PROGRAM POU
VAR
	
	A : BOOL := FALSE;
	B : BOOL := FALSE;
	C : BOOL := FALSE;
	D : BOOL := FALSE;

	TON_0: TON;
END_VAR

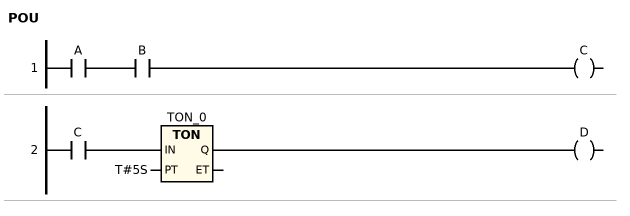
// NETWORK 1
C := A AND B;

// NETWORK 2
TON_0(IN := C, PT := T#5S); // TON
D := TON_0.Q;

END_PROGRAM

(* stored: Version 1.1.0.1, ProductVersion 3.1.4024.3
   POU POU: Id {ac75e950-3c46-48c7-b1a2-09646e49d2dd}, SpecialFunc None *)
